PROGRAM Trim_Saw_Pre
VAR
	tonSawEntryPhotoEye				: TON;
	tonSawExitPhotoEye				: TON;
	tonFootSwitch					: TON;
	lrBoardThickness				: ARRAY[0..1] OF LREAL;
END_VAR

tonSawEntryPhotoEye(IN := Inputs.i_xSawEntryPhotoEye, PT := T#50MS);
tonSawExitPhotoEye(IN := Inputs.i_xSawExitPhotoEye, PT := T#50MS);
tonFootSwitch(IN := Inputs.i_xFootSwitch, PT := T#50MS);

IF HMI.lrLaserScaling[0] <> 0 THEN
	lrBoardThickness[0] := Inputs.i_iBoardThickness[0] / HMI.lrLaserScaling[0] + HMI.lrLaserOffset[0];
	HMI.lrCurrentThickenss[0] := lrBoardThickness[0];
END_IF

IF HMI.lrLaserScaling[1] <> 0 THEN
	lrBoardThickness[1] := Inputs.i_iBoardThickness[1] / HMI.lrLaserScaling[1] + HMI.lrLaserOffset[1];
	HMI.lrCurrentThickenss[1] := lrBoardThickness[1];
END_IF

IF tonFootSwitch.Q THEN
	Outputs.q_xDeck3Stopper := TRUE;
ELSE
	Outputs.q_xDeck3Stopper := FALSE;
END_IF

IF HMI.xSlowFastButton THEN
	//Set conveyor speed to slow
ELSE
	//Set conveyor speed to fast
END_IF

//For Demo
//lrBoardThickness := HMI.lrCurrentThickenss;

IF tonSawEntryPhotoEye.Q THEN
	Inputs.i_xSawEntryPhotoEye := FALSE;
END_IF

IF tonSawExitPhotoEye.Q THEN
	Inputs.i_xSawExitPhotoEye := FALSE;
END_IF

END_PROGRAM

(* stored: Version 1.1.0.1, ProductVersion 3.1.4024.4
   POU Trim_Saw_Pre: Id {eee4eff6-bf88-4f1c-93f2-342fd6996b21}, SpecialFunc None *)
